Staubli VAL3: calcForce.pgx

public program calcForce(num& x_nDetectValue[], num& x_nFTValue[])
  local num l_nSequence
begin

  //通过Wacoh F/T Sensor Instruction Manual中的公式计算测得的力和力矩值

  //F/T Value=(detected value-zero point value)/main axis sensitivity
  for l_nSequence=0 to 5
    x_nFTValue[l_nSequence]=(x_nDetectValue[l_nSequence]-nZeroPoint[l_nSequence])/nSensitivity[l_nSequence]
    //x_nFTValue[l_nSequence]=(x_nDetectValue[l_nSequence]-8192)/nSensitivity[l_nSequence]
  endFor

end
